// TIA Portal V19 export
DATA_BLOCK "DBF_Safety"   // DB901, F_DB
{ S7_Optimized_Access := 'TRUE' }
// stored: AutoNumber false
   VAR
      TrueSafety { ExternalAccessible := 'False'; ExternalVisible := 'False'; ExternalWritable := 'False'} : Bool := TRUE;   // Safety Bool always TRUE
      FalseSafety { ExternalAccessible := 'False'; ExternalVisible := 'False'; ExternalWritable := 'False'} : Bool := FALSE;   // Safety Bool always FALSE
      Reset { ExternalAccessible := 'False'; ExternalVisible := 'False'; ExternalWritable := 'False'} : Bool;   // Reset bool
      ResetDoor { ExternalAccessible := 'False'; ExternalVisible := 'False'; ExternalWritable := 'False'} : Bool;   // Reset bool on maintenance door acces
      i_EStopOnMainCabinet { ExternalAccessible := 'False'; ExternalVisible := 'False'; ExternalWritable := 'False'} : Bool;   // Emergency stop state on main cabinet
      i_EStopLeftRopePull { ExternalAccessible := 'False'; ExternalVisible := 'False'; ExternalWritable := 'False'} : Bool;   // Emergency stop state rope pull left
      i_EStopRightRopePull { ExternalAccessible := 'False'; ExternalVisible := 'False'; ExternalWritable := 'False'} : Bool;   // Emergency stop state rope full right
      i_EStopEntryDoor { ExternalAccessible := 'False'; ExternalVisible := 'False'; ExternalWritable := 'False'} : Bool;   // Emergency stop state on entry guard locking
      i_DoorAcces { ExternalAccessible := 'False'; ExternalVisible := 'False'; ExternalWritable := 'False'} : Bool;   // Door state
      i_GateAccesCBS { ExternalAccessible := 'False'; ExternalVisible := 'False'; ExternalWritable := 'False'} : Bool;   // Gate acces state
      i_EStopControlRoom { ExternalAccessible := 'False'; ExternalVisible := 'False'; ExternalWritable := 'False'} : Bool;   // Emergency stop in the control room
      i_PedestrialDoorAcces { ExternalAccessible := 'False'; ExternalVisible := 'False'; ExternalWritable := 'False'} : Bool;   // Pedestrial door access state
      i_CaptiveKeyInLock { ExternalAccessible := 'False'; ExternalVisible := 'False'; ExternalWritable := 'False'} : Bool;   // Captive key on Lock
      i_EStopFromLeftRobot { ExternalAccessible := 'False'; ExternalVisible := 'False'; ExternalWritable := 'False'} : Bool;   // Emergency stop from flex pendant on the left robot
      i_EStopFromRightRobot { ExternalAccessible := 'False'; ExternalVisible := 'False'; ExternalWritable := 'False'} : Bool;   // Emergency stop from flex pendant on the right robot
      i_ReqEnableAirLeft { ExternalAccessible := 'False'; ExternalVisible := 'False'; ExternalWritable := 'False'} : Bool;   // Request enavle air pressure supply from left robot
      i_ReqEnableAirRight { ExternalAccessible := 'False'; ExternalVisible := 'False'; ExternalWritable := 'False'} : Bool;   // Request enavle air pressure supply from right robot
      i_RobotLeftStopped { ExternalAccessible := 'False'; ExternalVisible := 'False'; ExternalWritable := 'False'} : Bool;   // Left robot stooped
      i_RobotRightStopped { ExternalAccessible := 'False'; ExternalVisible := 'False'; ExternalWritable := 'False'} : Bool;   // Right robot stopped
      i_VacuumPumpRunning { ExternalAccessible := 'False'; ExternalVisible := 'False'; ExternalWritable := 'False'} : Bool;
      o_EnableAirSupplyLeftRobot { ExternalAccessible := 'False'; ExternalVisible := 'False'; ExternalWritable := 'False'} : Bool;   // Enable air pressure supply for left robot
      o_EnableAirSupplyRightRobot { ExternalAccessible := 'False'; ExternalVisible := 'False'; ExternalWritable := 'False'} : Bool;   // Enable air pressure supply for right robot
      o_EnableAirSupplySuctionUnit { ExternalAccessible := 'False'; ExternalVisible := 'False'; ExternalWritable := 'False'} : Bool;   // Enable air pressure supply for suction unit
      o_EStopSuctionUnit { ExternalAccessible := 'False'; ExternalVisible := 'False'; ExternalWritable := 'False'} : Bool;   // Emergency stop state to suction unit
      o_EStopToLeftRobot { ExternalAccessible := 'False'; ExternalVisible := 'False'; ExternalWritable := 'False'} : Bool;   // Cell emergency stop to left robot
      o_EStopToRightRobot { ExternalAccessible := 'False'; ExternalVisible := 'False'; ExternalWritable := 'False'} : Bool;   // Cell emergency stop to right robot
      o_OperatorProtectionToLeftRobot { ExternalAccessible := 'False'; ExternalVisible := 'False'; ExternalWritable := 'False'} : Bool;   // Operator protection state to the left robot
      o_OperatorProtectionToRightRobot { ExternalAccessible := 'False'; ExternalVisible := 'False'; ExternalWritable := 'False'} : Bool;   // Operator protection state to the right robot
      o_VacuumRunningDelayed { ExternalAccessible := 'False'; ExternalVisible := 'False'; ExternalWritable := 'False'} : Bool;   // Vacuum running delayed of
      l_GlobalEmergencyStopCell { ExternalAccessible := 'False'; ExternalVisible := 'False'; ExternalWritable := 'False'} : Bool;   // Global Emergency stop cell state
      l_GlobalEmergencyStop { ExternalAccessible := 'False'; ExternalVisible := 'False'; ExternalWritable := 'False'} : Bool;   // Global Emergency stop state
      l_GlobalEStopToLeftRobot { ExternalAccessible := 'False'; ExternalVisible := 'False'; ExternalWritable := 'False'} : Bool;   // Global Emergency stop state send to left robot
      l_GlobalEStopToRightRobot { ExternalAccessible := 'False'; ExternalVisible := 'False'; ExternalWritable := 'False'} : Bool;   // Global Emergency stop state send to right robot
      l_GlobalOperatorProtection { ExternalAccessible := 'False'; ExternalVisible := 'False'; ExternalWritable := 'False'} : Bool;   // Global door and gate state
      xErrorReadFromLeft { ExternalAccessible := 'False'; ExternalVisible := 'False'; ExternalWritable := 'False'} : Bool;
      xErrorReadFromRight { ExternalAccessible := 'False'; ExternalVisible := 'False'; ExternalWritable := 'False'} : Bool;
      xErrorWriteToLeft { ExternalAccessible := 'False'; ExternalVisible := 'False'; ExternalWritable := 'False'} : Bool;
      xErrorWriteToRight { ExternalAccessible := 'False'; ExternalVisible := 'False'; ExternalWritable := 'False'} : Bool;
      xAuthorStart { ExternalAccessible := 'False'; ExternalVisible := 'False'; ExternalWritable := 'False'} : Bool;
      xVacuumPumpRunning { ExternalAccessible := 'False'; ExternalVisible := 'False'; ExternalWritable := 'False'} : Bool;
   END_VAR
BEGIN
END_DATA_BLOCK
